FUNCTION_BLOCK EM_Transport_Mechanische_Stop EXTENDS EM_Transport IMPLEMENTS ITF_EM_Transport_Mechanische_Stop

VAR
	fbMechanischeStop_mem : STRUCT_EM_Mechanische_Stop;
	Klep		: CM_Valve;
END_VAR

(*
$$$$$$$$\                                                                   $$\       $$$$$$$$\                     $$\                                         $$\                     
$$  _____|                                                                  $$ |      $$  _____|                    \__|                                        \__|                    
$$ |   $$$$$$\   $$$$$$\  $$$$$$$\  $$\  $$\  $$\  $$$$$$\   $$$$$$\   $$$$$$$ |      $$ |      $$$$$$$\   $$$$$$\  $$\ $$$$$$$\   $$$$$$\   $$$$$$\   $$$$$$\  $$\ $$$$$$$\   $$$$$$\  
$$$$$\ \____$$\ $$  __$$\ $$  __$$\ $$ | $$ | $$ |$$  __$$\ $$  __$$\ $$  __$$ |      $$$$$\    $$  __$$\ $$  __$$\ $$ |$$  __$$\ $$  __$$\ $$  __$$\ $$  __$$\ $$ |$$  __$$\ $$  __$$\ 
$$  __|$$$$$$$ |$$ |  \__|$$ |  $$ |$$ | $$ | $$ |$$ /  $$ |$$ /  $$ |$$ /  $$ |      $$  __|   $$ |  $$ |$$ /  $$ |$$ |$$ |  $$ |$$$$$$$$ |$$$$$$$$ |$$ |  \__|$$ |$$ |  $$ |$$ /  $$ |
$$ |  $$  __$$ |$$ |      $$ |  $$ |$$ | $$ | $$ |$$ |  $$ |$$ |  $$ |$$ |  $$ |      $$ |      $$ |  $$ |$$ |  $$ |$$ |$$ |  $$ |$$   ____|$$   ____|$$ |      $$ |$$ |  $$ |$$ |  $$ |
$$ |  \$$$$$$$ |$$ |      $$ |  $$ |\$$$$$\$$$$  |\$$$$$$  |\$$$$$$  |\$$$$$$$ |      $$$$$$$$\ $$ |  $$ |\$$$$$$$ |$$ |$$ |  $$ |\$$$$$$$\ \$$$$$$$\ $$ |      $$ |$$ |  $$ |\$$$$$$$ |
\__|   \_______|\__|      \__|  \__| \_____\____/  \______/  \______/  \_______|      \________|\__|  \__| \____$$ |\__|\__|  \__| \_______| \_______|\__|      \__|\__|  \__| \____$$ |
                                                                                                          $$\   $$ |                                                          $$\   $$ |
                                                                                                          \$$$$$$  |                                                          \$$$$$$  |
                                                                                                           \______/                                                            \______/ 
*)

//********************************Init***********************************
Klep();
SUPER^();
										
//********************************ZEROING***********************************	
(*								
fb_mem.STS.Auto 			:= FALSE;
fb_mem.STS.Manueel 			:= FALSE;
fb_mem.STS.Starting_SC 		:= FALSE;
fb_mem.STS.Execute_SC 		:= FALSE;
fb_mem.STS.Resetting_SC 	:= FALSE;
fb_mem.STS.Holding_SC 		:= FALSE;
fb_mem.STS.Unholding_SC 	:= FALSE;
fb_mem.STS.Suspending_SC 	:= FALSE;
fb_mem.STS.Unsuspending_SC 	:= FALSE;
fb_mem.STS.Aborting_SC 		:= FALSE;
fb_mem.STS.Clearing_SC 		:= FALSE;
fb_mem.STS.Stopping_SC 		:= FALSE;
fb_mem.STS.Completing_SC 	:= FALSE;
*)

//********************************Auto manual logic***********************************


//********************************Exeptionhandling***********************************

//********************************Action case***********************************


//********************************ZEROING***********************************
//Control Signals 
(*
fb_mem.CS.Auto            := FALSE;
fb_mem.CS.Manueel         := FALSE;
fb_mem.CS.Start           := FALSE;
fb_mem.CS.Stop            := FALSE;
fb_mem.CS.Reset           := FALSE;
fb_mem.CS.Abort           := FALSE;
fb_mem.CS.Clear           := FALSE;
fb_mem.CS.UnSuspend       := FALSE;
fb_mem.CS.Suspend         := FALSE;
fb_mem.CS.UnHold          := FALSE;
fb_mem.CS.Hold            := FALSE;
*)

{warning 'add method implementation '}
METHOD Close : BOOL
END_METHOD

{warning 'add method implementation '}
METHOD Open : BOOL
END_METHOD

PROPERTY Stop_State : E_Mechanische_Stop
GET
Stop_State := fbMechanischeStop_mem.STS.State;
END_GET
END_PROPERTY

{warning 'add method implementation '}
METHOD ZeroAllValues : BOOL
END_METHOD

END_FUNCTION_BLOCK

(* stored: Version 1.1.0.1, ProductVersion 3.1.4024.12
   POU EM_Transport_Mechanische_Stop: Id {b7168c61-ecd4-4685-b920-755ca0b861b8}, SpecialFunc None
   Folder Methods: Id {3d8b66f8-3d7c-495b-80c7-324b66a87557}
   Folder Properties: Id {9e87a29a-b81d-42a4-ad34-326d6677771f}
   Method Close: Id {bc7183c4-aedc-4363-8e85-1e5ded2c28c9}
   Method Open: Id {1e494ea6-65cf-4ee9-9f18-11ad53317a66}
   Property Stop_State: Id {3694e7d8-987e-4d1e-8f5d-02e4bf119952}
   Get Get: Id {e0e286d6-582b-4de6-8651-08ea60a23a4d}
   Method ZeroAllValues: Id {89462386-6c82-4719-9f6c-5c50a1373597} *)
